// IEEE-754 classification by integer exponent bits; no floating-point operation.
// Safe with runtime floating-point exceptions enabled, including signaling NaNs.
FUNCTION F_IsFiniteReal : BOOL
VAR_INPUT value : REAL; END_VAR
VAR bits : DWORD; END_VAR

Tc2_System.MEMCPY(destAddr := ADR(bits), srcAddr := ADR(value), n := SIZEOF(bits));
F_IsFiniteReal := (bits AND DWORD#16#7F800000) <> DWORD#16#7F800000;

END_FUNCTION

(* stored: Version 1.1.0.1
   POU F_IsFiniteReal: Id {be6c918e-2b14-4e17-8b0e-cf8c082c3118} *)
